SUBAPPLICATION CONCAT_WSTRING (* Subapplication Type *)
  (* Standard: 61499-2 *)
  (* Version 1.0, 2023-04-10, derPi *)
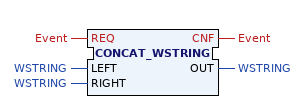
  EVENT_INPUT
    REQ; (* Normal Execution Request *)
  END_EVENT
  EVENT_OUTPUT
    CNF; (* Execution Confirmation *)
  END_EVENT
  VAR_INPUT
    LEFT : WSTRING;
    RIGHT : WSTRING;
  END_VAR
  VAR_OUTPUT
    OUT : WSTRING;
  END_VAR
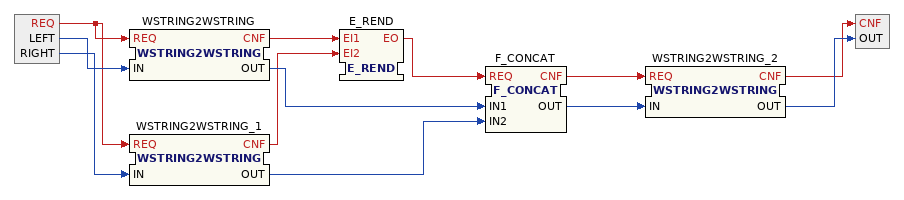
  FBS
    WSTRING2WSTRING : WSTRING2WSTRING;
    WSTRING2WSTRING_1 : WSTRING2WSTRING;
    F_CONCAT : F_CONCAT;
    E_REND : E_REND;
    WSTRING2WSTRING_2 : WSTRING2WSTRING;
  END_FBS
  EVENT_CONNECTIONS
    WSTRING2WSTRING.CNF TO E_REND.EI1;
    WSTRING2WSTRING_1.CNF TO E_REND.EI2;
    E_REND.EO TO F_CONCAT.REQ;
    REQ TO WSTRING2WSTRING.REQ;
    REQ TO WSTRING2WSTRING_1.REQ;
    F_CONCAT.CNF TO WSTRING2WSTRING_2.REQ;
    WSTRING2WSTRING_2.CNF TO CNF;
  END_CONNECTIONS
  DATA_CONNECTIONS
    WSTRING2WSTRING.OUT TO F_CONCAT.IN1;
    WSTRING2WSTRING_1.OUT TO F_CONCAT.IN2;
    LEFT TO WSTRING2WSTRING.IN;
    RIGHT TO WSTRING2WSTRING_1.IN;
    F_CONCAT.OUT TO WSTRING2WSTRING_2.IN;
    WSTRING2WSTRING_2.OUT TO OUT;
  END_CONNECTIONS
END_SUBAPPLICATION
